(*
SPDX-FileCopyrightText: © 2026 Oleksandr Tiutyk <trofimich@gmail.com>
SPDX-License-Identifier: MIT
License: https://opensource.org/license/mit
*)

INTERFACE IWaitAndPickActivity EXTENDS IExclusiveCompositeActivity

METHOD AddBarnch : DINT
VAR_INPUT
	condition : ICondition;
	activity : IActivity;
END_VAR
END_METHOD

{attribute 'monitoring' := 'call'}
PROPERTY FINAL CurrentActivity : IActivity
GET
END_GET
END_PROPERTY

{attribute 'monitoring' := 'call'}
PROPERTY FINAL CurrentBranchIndex : DINT
GET
END_GET
END_PROPERTY

END_INTERFACE

(* stored: Version 1.1.0.1
   Itf IWaitAndPickActivity: Id {7c324977-e60a-45fb-9360-b0ea3e5e5a57}
   Method AddBarnch: Id {cceb521c-fa78-4662-bb9f-0d9fd6a8e81a}
   Property CurrentActivity: Id {bb402ee2-2866-4ba0-9ad2-a370ad0e4104}
   Get Get: Id {b705ff2e-5341-48ec-ab21-7fbc8de677f7}
   Property CurrentBranchIndex: Id {32f18dd6-a162-4250-9243-ea54bc3d502c}
   Get Get: Id {d27bf5f9-7556-466e-82b0-91ec1d21094c} *)
